FUNCTION_BLOCK DigitalInput_DebounceFallingEdge EXTENDS CyclicComponent IMPLEMENTS I_DigitalInput
VAR
	Input : I_DigitalInput;
	{attribute 'hide'}
	_DebounceTime		: TIME;
	DebounceFallingEdge : TOF;
END_VAR

METHOD CyclicLogic
DebounceFallingEdge(IN := Input.IsActive, PT := _DebounceTime);
END_METHOD

{attribute 'monitoring' := 'call'}
PROPERTY DebounceTime : TIME
GET
DebounceTime := _DebounceTime;
END_GET
SET
_DebounceTime := DebounceTime;
END_SET
END_PROPERTY

(*FB_Init is always available implicitly and it is used primarily for initialization.
The return value is not evaluated. For a specific influence, you can also declare the
methods explicitly and provide additional code there with the standard initialization
code. You can evaluate the return value.*)
METHOD FB_Init : BOOL
VAR_INPUT
	(* TRUE: the retain variables are initialized (reset warm / reset cold)*)
	bInitRetains : BOOL;

	(* TRUE: the instance will be copied to the copy code afterward (online change)   *)
	bInCopyCode : BOOL;
	Name		: T_MaxString;
	Input		: I_DigitalInput;
END_VAR
THIS^.Input := Input;
END_METHOD

{attribute 'monitoring' := 'call'}
PROPERTY Force : E_ForceState
GET
Force := Input.Force;
END_GET
SET
Input.Force := Force;
END_SET
END_PROPERTY

{attribute 'monitoring' := 'call'}
PROPERTY IsActive : BOOL
GET
IsActive := DebounceFallingEdge.Q;
END_GET
END_PROPERTY

END_FUNCTION_BLOCK

(* stored: Version 1.1.0.1, ProductVersion 3.1.4026.18
   POU DigitalInput_DebounceFallingEdge: Id {083cf1be-1e7e-46ce-bfd5-ad7ee3eb164b}, SpecialFunc None
   Method CyclicLogic: Id {ae2942a5-4ed7-42cf-a4cb-e042cd871c00}
   Property DebounceTime: Id {d155dacc-cab3-40eb-b482-dad21e9c6f3c}
   Get Get: Id {7972a916-6c45-4472-ae12-a9a3950d5fb8}
   Set Set: Id {5c3281f8-a39d-418c-9c3a-0e6800aa1523}
   Method FB_Init: Id {1e8097b5-11f4-4040-bd2b-e892d00d9ccc}
   Property Force: Id {59c1549a-25dc-4145-a4d5-e3681b484a1f}
   Get Get: Id {d93ff538-c535-4e54-b785-26bc0890559a}
   Set Set: Id {2c07069c-f60d-4ee0-b5ce-6bb6f350ab78}
   Property IsActive: Id {79f07904-9f38-4600-8964-2ee70ac3658a}
   Get Get: Id {8ee02001-ba05-4051-b35a-909370dad754} *)
